Fanuc KAREL source: print_line.kl

PROGRAM print_line
%NOBUSYLAMP
%NOLOCKGROUP

VAR
	str : STRING[32]
%from tpe.klh %import get_string_arg
%from display.klh %import print_line

BEGIN
	str = tpe__get_string_arg(1)
	display__print_line(str)
END print_line
